TYPE "JB_WeldingSetUp"
VERSION : 0.1
// Block: JB_WeldingSetUp
   STRUCT
      MaterialWidth : LReal;
      MeasureSheetEdgeReference : LReal;
      WeldingDirection : Bool;
      CorrStartWelding : LReal;
      CorrStopWelding : LReal;
   END_STRUCT;

END_TYPE
